FUNCTION_BLOCK AxesManager
VAR_INPUT
END_VAR
VAR_OUTPUT
	// am Punkt angekommen
	bPunktAngefahren: BOOL;
END_VAR
VAR
	// Achsen der Maschine (X-Z-Achse)
	xAchse: AXIS_REF;
	zAchse: AXIS_REF;
	
	stPunkt: ST_2DPoint;
	
	// MC2 Funktionen
	fbAxisPowerX: MC_Power;
	fbAxisMoveX: MC_MoveAbsolute;
	
	fbAxisPowerZ: MC_Power;
	fbAxisMoveZ: MC_MoveAbsolute;
	
	// Velocity
	xVelo: LREAL := 100;
	zVelo: LREAL := 100;
	
	bMoveAxes: BOOL := FALSE;
	
	bXMoved: BOOL := FALSE;
	bZMoved: BOOL := FALSE;
END_VAR

xAchse.ReadStatus();
zAchse.ReadStatus();

fbAxisMoveX(Axis := xAchse, Velocity := xVelo, Execute := bMoveAxes, Position := stPunkt.x, Done => bXMoved);
fbAxisMoveZ(Axis := zAchse, Velocity := zVelo, Execute := bMoveAxes, Position := stPunkt.y, Done => bZMoved);

bPunktAngefahren := bXMoved AND bZMoved;

PROPERTY PUBLIC CurrentPoint : REFERENCE TO ST_2DPoint
GET
CurrentPoint REF= stPunkt;
END_GET
END_PROPERTY

METHOD PUBLIC Enable : BOOL
VAR_INPUT
	bEnableAxes: BOOL;
END_VAR
fbAxisPowerX(Axis := xAchse, Enable := bEnableAxes, Enable_Positive := bEnableAxes, Enable_Negative := bEnableAxes);
fbAxisPowerZ(Axis := zAchse, Enable := bEnableAxes, Enable_Positive := bEnableAxes, Enable_Negative := bEnableAxes);
END_METHOD

METHOD PUBLIC LogAxes : BOOL
VAR_INPUT
END_VAR
ADSLOGLREAL(
	msgCtrlMask := ADSLOG_MSGTYPE_HINT,
	msgFmtStr := 'x-Achse: %f',
	lrealArg := xAchse.NcToPlc.ActPos
);

ADSLOGLREAL(
	msgCtrlMask := ADSLOG_MSGTYPE_HINT,
	msgFmtStr := 'z-Achse: %f',
	lrealArg := zAchse.NcToPlc.ActPos
);
END_METHOD

METHOD PUBLIC Start : BOOL
VAR_INPUT
	stPunkt: REFERENCE TO ST_2DPoint;
END_VAR
THIS^.stPunkt := stPunkt;
bMoveAxes := TRUE;
END_METHOD

METHOD PUBLIC Stop : BOOL
VAR_INPUT
END_VAR
bMoveAxes := FALSE;
END_METHOD

END_FUNCTION_BLOCK

(* stored: Version 1.1.0.1, ProductVersion 3.1.4024.3
   POU AxesManager: Id {2d19b545-a977-41d5-ac65-a00e41c4aca4}, SpecialFunc None
   Property CurrentPoint: Id {2b66fb39-4ec5-4378-86d6-44900e4437d7}
   Get Get: Id {cef1edba-712b-497b-8d21-4187a65ea703}
   Method Enable: Id {9967a336-49b9-4a03-ba39-133db437a907}
   Method LogAxes: Id {e9378cc9-a699-4554-a902-db82d5906abc}
   Method Start: Id {1cafe01f-d4a8-4712-a211-1a5b246bb457}
   Method Stop: Id {e20ac144-d3a4-463f-bfe5-2ec53d758fbe} *)
